PROGRAM P92_Maintenance
VAR_INPUT
	bBuzzerStop				: BOOL;
	nCaseSignalTower		: INT;
END_VAR
VAR_OUTPUT

END_VAR
VAR
	(* Input *)
	//Light
	bLightCP				: BOOL;
	rTrigReactorCabinetSwitch	: R_TRIG;
	rTrigReactorCabinetMagnet 	: R_TRIG;
	fTrigReactorCabinetMagnet 	: F_TRIG;
	rTrigGasCabinetSwitch		: R_TRIG;
	rTrigGasCabinetMagnet		: R_TRIG;
	fTrigGasCabinetMagnet		: F_TRIG;

	bReactorCabinetLampSwitch : BOOL;
	bGasCabinetLampSwitch	: BOOL;
	
	bReactorCabientMagnet	: BOOL;
	bGasCabinetMagnet		: BOOL;
	bPowerDistributeMagnet	: BOOL;
	
	(* Output to Device *)
	// Cabinet Lamp
	bReactorCabinetLamp		: BOOL;
	bGasCabinetLamp			: BOOL;
	bPowerDistributeLamp	: BOOL;
	
	bSMPS24V480WFault		: BOOL;
	bSMPS24V72WFault		: BOOL;
	bSMPS15VPlusFault		: BOOL;
	bSMPS15VMinusFault		: BOOL;
	bSMPS15CP				: BOOL;
	// Signal Tower
	bSignalTower			: BYTE;
	TimerSignalTower		: TON;
END_VAR

(* Read from Device Value *)
//Lamp
bLightCP 				:= GVL_IO.aDigitalInputIO[5].6;
bReactorCabientMagnet 	:= GVL_IO.aDigitalInputIO[3].6;
bGasCabinetMagnet 		:= GVL_IO.aDigitalInputIO[3].7;
bPowerDistributeMagnet	:= GVL_IO.aDigitalInputIO[4].0;

bSMPS15CP				:= GVL_IO.aDigitalInputIO[5].7;
//SMPS
bSMPS24V480WFault	:= NOT(GVL_IO.aDigitalInputIO[4].3);
bSMPS24V72WFault	:= NOT(GVL_IO.aDigitalInputIO[4].4);
bSMPS15VPlusFault	:= NOT(GVL_IO.aDigitalInputIO[4].5);
bSMPS15VMinusFault	:= NOT(GVL_IO.aDigitalInputIO[4].6);

// Reactor Cabinet Lamp
rTrigReactorCabinetSwitch(CLK:=GVL_IO.aDigitalInputIO[1].2);
rTrigReactorCabinetMagnet(CLK:=GVL_IO.aDigitalInputIO[3].6);
fTrigReactorCabinetMagnet(CLK:=GVL_IO.aDigitalInputIO[3].6);
IF rTrigReactorCabinetSwitch.Q OR rTrigReactorCabinetMagnet.Q OR fTrigReactorCabinetMagnet.Q THEN
	bReactorCabinetLamp := NOT(bReactorCabinetLamp);
END_IF
// Gas Delivery Cabinet Lamp
rTrigGasCabinetSwitch(CLK:= GVL_IO.aDigitalInputIO[1].3);
rTrigGasCabinetMagnet(CLK:= GVL_IO.aDigitalInputIO[3].7);
fTrigGasCabinetMagnet(CLK:= GVL_IO.aDigitalInputIO[3].7);
IF rTrigGasCabinetSwitch.Q THEN
	bGasCabinetLamp := NOT(bGasCabinetLamp);
ELSIF fTrigGasCabinetMagnet.Q THEN
	bGasCabinetLamp := TRUE;
ELSIF rTrigGasCabinetMagnet.Q THEN
	bGasCabinetLamp := FALSE;
END_IF
// Power Distribute Unit Lamp
bPowerDistributeLamp := NOT(bPowerDistributeMagnet); //Magnet Switch

(* Blink Signal Tower *)
CASE nCaseSignalTower OF
	1: //RED 
		TimerSignalTower(IN:=TRUE, PT:=T#500MS);
		IF TimerSignalTower.Q THEN
			TimerSignalTower(IN:=FALSE);
			IF bSignalTower = 0 THEN
				bSignalTower := 2#0000_0001; // RED
			ELSE
				bSignalTower := 0;
			END_IF
		END_IF
	2: //YELLOW 
		TimerSignalTower(IN:=TRUE, PT:=T#1S);
		IF TimerSignalTower.Q THEN
			TimerSignalTower(IN:=FALSE);
			IF bSignalTower = 0 THEN
				bSignalTower := 2#0000_0010; // YELLOW
			ELSE
				bSignalTower := 0;
			END_IF
		END_IF
	3: //GREEN
		bSignalTower := 2#0000_0100;
	4: //BLUE
		bSignalTower := 2#0000_1000;
	5: //WHITE
		bSignalTower := 2#0001_0000;
	6: //BUZZER
		bSignalTower := 2#0010_0001;
		IF bBuzzerStop THEN
			bSignalTower := 2#0000_0001;
		END_IF
	ELSE
		bSignalTower := 0;
END_CASE

(* Write to Device Value *)
GVL_IO.aDigitalOutputIO[2].5 	:= bReactorCabinetLamp;
GVL_IO.aDigitalOutputIO[2].6 	:= bGasCabinetLamp;
GVL_IO.aDigitalOutputIO[2].7 	:= bPowerDistributeLamp;

//SignalTower
GVL_IO.aDigitalOutputIO[1].0 		:= bSignalTower.0; //0:RED-Alarm,
GVL_IO.aDigitalOutputIO[1].1 		:= bSignalTower.1; //1:YELLOW,-Warning 
GVL_IO.aDigitalOutputIO[1].2 		:= bSignalTower.2; //2:GREEN-Running
GVL_IO.aDigitalOutputIO[1].3 		:= bSignalTower.3; //3:BLUE-Idle
GVL_IO.aDigitalOutputIO[1].4 		:= bSignalTower.4; //4:WHITE-Maint
GVL_IO.aDigitalOutputIO[1].5 		:= bSignalTower.5; //5:BUZZER-Alarm

END_PROGRAM

(* stored: Version 1.1.0.1, ProductVersion 3.1.4026.11
   POU P92_Maintenance: Id {17478ea4-373a-4676-aa4e-f86e85a19514}, SpecialFunc None *)
